// TIA Portal V16 export
// export: Created 2022-11-17T15:49:45.6262472Z, ExportSetting WithDefaults, DisplayName Totally Integrated Automation Portal, DisplayVersion V16 Update 6, DisplayName TIA Portal Version Control Interface, DisplayVersion V16 Update 2, DisplayName TIA Portal Openness, DisplayVersion V16 Update 6, DisplayName SINAMICS Startdrive Advanced, DisplayVersion V16 Update 5, DisplayName SINAMICS Startdrive G130, G150, S120, S150, SINAMICS MV, S210, DisplayVersion V16 Update 5, DisplayName SINAMICS Startdrive G110M, G120, G120C, G120D, G120P, G115D, DisplayVersion V16 Update 5, DisplayName STEP 7 Professional, DisplayVersion V16 Update 6, DisplayName STEP 7 Safety, DisplayVersion V16, DisplayName WinCC Advanced, DisplayVersion V16 Update 6
DATA_BLOCK "DB246_Program4"   // DB246
{ S7_Optimized_Access := 'FALSE' }
AUTHOR : Robopac
VERSION : 0.0
// stored: AutoNumber false, IsOnlyStoredInLoadMemory false, IsWriteProtectedInAS false
   VAR RETAIN
      Program4 { S7_SetPoint := 'True'} : "DatiProgramma";
   END_VAR
BEGIN
   Program4.Wrapping := TRUE;
   Program4.TopLenght := 500;
   Program4.TopRelease := 0;
   Program4.TopDown := 0;
   Program4.Top := 4;
   Program4.PressurePTime := 0;
   Program4.LifterTime := 0;
   Program4.RevOverContrast := 1;
   Program4.RopeEndCycle := 16#02;
   Program4.Spare4 := 16#01;
   Program4.RopeTime := 1500;
   Program4.RevOverClamp := 1;
   Program4.FilmForceFinalRev := 10;
   Program4.FilmPrestretchFinalRev := 100;
   Program4.ArmSpeed := 100;
   Program4.CarriageDown4Top := 500;
   Program4.TopDownTime := 1500;
   Program4.LapsUnderTop := 0;
   Program4.Spare6 := 0;
   Program4.Spare7 := 0;
   Program4.Spare8 := 0;
   Program4.Spare9 := 0;
   Program4.Spare10 := 0;
   Program4.Spare11 := 0;
   Program4.Spare12 := 0;
   Program4.Overlap0_1 := 0;
   Program4.Height1 := 130;
   Program4.Landmark1 := FALSE;
   Program4.Lifter1 := FALSE;
   Program4.SpareBit1H1 := FALSE;
   Program4.Airblower1 := TRUE;
   Program4.NextStep1 := TRUE;
   Program4.PressureP1 := TRUE;
   Program4.SpareByte2H1 := 16#00;
   Program4.Revolution1 := 1;
   Program4.RopeUnit1_1 := 16#01;
   Program4.RopeUnit1_2 := 16#01;
   Program4.FilmForce1 := 5;
   Program4.FilmPrestretch1 := 200;
   Program4.Spare3H1 := 0;
   Program4.Spare49 := 0;
   Program4.Spare50 := 0;
   Program4.Spare51 := 0;
   Program4.Spare52 := 0;
   Program4.Spare53 := 0;
   Program4.Overlap1_2 := 0;
   Program4.Height2 := 50;
   Program4.Landmark2 := FALSE;
   Program4.Lifter2 := FALSE;
   Program4.SpareBit1H2 := FALSE;
   Program4.Airblower2 := TRUE;
   Program4.NextStep2 := TRUE;
   Program4.PressureP2 := TRUE;
   Program4.SpareByte2H2 := 16#00;
   Program4.Revolution2 := 1;
   Program4.RopeUnit2_1 := 16#01;
   Program4.RopeUnit2_2 := 16#01;
   Program4.FilmForce2 := 20;
   Program4.FilmPrestretch2 := 200;
   Program4.Spare3H2 := 0;
   Program4.Spare54 := 0;
   Program4.Spare55 := 0;
   Program4.Spare56 := 0;
   Program4.Spare57 := 0;
   Program4.Spare58 := 0;
   Program4.Overlap2_3 := 100;
   Program4.Height3 := -50;
   Program4.Landmark3 := TRUE;
   Program4.Lifter3 := FALSE;
   Program4.SpareBit1H3 := FALSE;
   Program4.Airblower3 := TRUE;
   Program4.NextStep3 := TRUE;
   Program4.PressureP3 := TRUE;
   Program4.SpareByte2H3 := 16#00;
   Program4.Revolution3 := 2;
   Program4.RopeUnit3_1 := 16#01;
   Program4.RopeUnit3_2 := 16#01;
   Program4.FilmForce3 := 30;
   Program4.FilmPrestretch3 := 200;
   Program4.Spare3H3 := 0;
   Program4.Spare59 := 0;
   Program4.Spare60 := 0;
   Program4.Spare61 := 380;
   Program4.Spare62 := 2800;
   Program4.Spare63 := 0;
   Program4.Overlap3_4 := 100;
   Program4.Height4 := 100;
   Program4.Landmark4 := FALSE;
   Program4.Lifter4 := FALSE;
   Program4.SpareBit1H4 := FALSE;
   Program4.Airblower4 := TRUE;
   Program4.NextStep4 := TRUE;
   Program4.PressureP4 := TRUE;
   Program4.SpareByte2H4 := 16#00;
   Program4.Revolution4 := 3;
   Program4.RopeUnit4_1 := 16#02;
   Program4.RopeUnit4_2 := 16#02;
   Program4.FilmForce4 := 30;
   Program4.FilmPrestretch4 := 200;
   Program4.Spare3H4 := 0;
   Program4.Spare64 := 0;
   Program4.Spare65 := 0;
   Program4.Spare66 := 0;
   Program4.Spare67 := 0;
   Program4.Spare68 := 0;
   Program4.Overlap4_5 := 0;
   Program4.Height5 := 50;
   Program4.Landmark5 := FALSE;
   Program4.Lifter5 := FALSE;
   Program4.SpareBit1H5 := FALSE;
   Program4.Airblower5 := TRUE;
   Program4.NextStep5 := FALSE;
   Program4.PressureP5 := FALSE;
   Program4.SpareByte2H5 := 16#00;
   Program4.Revolution5 := 1;
   Program4.RopeUnit5_1 := 16#01;
   Program4.RopeUnit5_2 := 16#01;
   Program4.FilmForce5 := 30;
   Program4.FilmPrestretch5 := 200;
   Program4.Spare3H5 := 0;
   Program4.Spare69 := 0;
   Program4.Spare70 := 0;
   Program4.Spare71 := 0;
   Program4.Spare72 := 0;
   Program4.Spare73 := 0;
   Program4.Overlap5_6 := 100;
   Program4.Height6 := 50;
   Program4.Landmark6 := FALSE;
   Program4.Lifter6 := FALSE;
   Program4.SpareBit1H6 := FALSE;
   Program4.Airblower6 := TRUE;
   Program4.NextStep6 := FALSE;
   Program4.PressureP6 := FALSE;
   Program4.SpareByte2H6 := 16#00;
   Program4.Revolution6 := 2;
   Program4.RopeUnit6_1 := 16#02;
   Program4.RopeUnit6_2 := 16#01;
   Program4.FilmForce6 := 20;
   Program4.FilmPrestretch6 := 200;
   Program4.Spare3H6 := 0;
   Program4.Spare74 := 0;
   Program4.Spare75 := 0;
   Program4.Spare76 := 0;
   Program4.Spare77 := 0;
   Program4.Spare78 := 0;
   Program4.Overlap6_7 := 0;
   Program4.Height7 := 0;
   Program4.Landmark7 := FALSE;
   Program4.Lifter7 := FALSE;
   Program4.SpareBit1H7 := FALSE;
   Program4.Airblower7 := FALSE;
   Program4.NextStep7 := TRUE;
   Program4.PressureP7 := FALSE;
   Program4.SpareByte2H7 := 16#00;
   Program4.Revolution7 := 1;
   Program4.RopeUnit7_1 := 16#01;
   Program4.RopeUnit7_2 := 16#01;
   Program4.FilmForce7 := 0;
   Program4.FilmPrestretch7 := 100;
   Program4.Spare3H7 := 0;
   Program4.Spare79 := 0;
   Program4.Spare80 := 0;
   Program4.Spare81 := 0;
   Program4.Spare82 := 0;
   Program4.Spare83 := 0;
   Program4.Overlap7_8 := 0;
   Program4.Height8 := 0;
   Program4.Landmark8 := FALSE;
   Program4.Lifter8 := FALSE;
   Program4.SpareBit1H8 := FALSE;
   Program4.Airblower8 := FALSE;
   Program4.NextStep8 := TRUE;
   Program4.PressureP8 := FALSE;
   Program4.SpareByte2H8 := 16#00;
   Program4.Revolution8 := 1;
   Program4.RopeUnit8_1 := 16#01;
   Program4.RopeUnit8_2 := 16#01;
   Program4.FilmForce8 := 0;
   Program4.FilmPrestretch8 := 100;
   Program4.Spare3H8 := 0;
   Program4.Spare84 := 0;
   Program4.Spare85 := 0;
   Program4.Spare86 := 0;
   Program4.Spare87 := 0;
   Program4.Spare88 := 0;
   Program4.Overlap8_9 := 0;
   Program4.Height9 := 0;
   Program4.Landmark9 := FALSE;
   Program4.Lifter9 := FALSE;
   Program4.SpareBit1H9 := FALSE;
   Program4.Airblower9 := FALSE;
   Program4.NextStep9 := TRUE;
   Program4.PressureP9 := FALSE;
   Program4.SpareByte2H9 := 16#00;
   Program4.Revolution9 := 1;
   Program4.RopeUnit9_1 := 16#01;
   Program4.RopeUnit9_2 := 16#01;
   Program4.FilmForce9 := 0;
   Program4.FilmPrestretch9 := 100;
   Program4.Spare3H9 := 0;
   Program4.Spare89 := 0;
   Program4.Spare90 := 0;
   Program4.Spare91 := 0;
   Program4.Spare92 := 0;
   Program4.Spare93 := 0;
   Program4.Overlap9_10 := 0;
   Program4.Height10 := 0;
   Program4.Landmark10 := FALSE;
   Program4.Lifter10 := FALSE;
   Program4.SpareBit1H10 := FALSE;
   Program4.Airblower10 := FALSE;
   Program4.NextStep10 := FALSE;
   Program4.PressureP10 := FALSE;
   Program4.SpareByte2H10 := 16#00;
   Program4.Revolution10 := 1;
   Program4.RopeUnit10_1 := 16#01;
   Program4.RopeUnit10_2 := 16#01;
   Program4.FilmForce10 := 0;
   Program4.FilmPrestretch10 := 100;
   Program4.Spare3H10 := 0;
   Program4.Spare94 := 0;
   Program4.Spare95 := 0;
   Program4.Spare96 := 0;
   Program4.Spare97 := 0;
   Program4.Spare98 := 0;
   Program4.Overlap10_11 := 0;
   Program4.Height11 := 0;
   Program4.Landmark11 := FALSE;
   Program4.Lifter11 := FALSE;
   Program4.SpareBit1H11 := FALSE;
   Program4.Airblower11 := FALSE;
   Program4.NextStep11 := TRUE;
   Program4.PressureP11 := FALSE;
   Program4.SpareByte2H11 := 16#00;
   Program4.Revolution11 := 1;
   Program4.RopeUnit11_1 := 16#01;
   Program4.RopeUnit11_2 := 16#01;
   Program4.FilmForce11 := 0;
   Program4.FilmPrestretch11 := 100;
   Program4.Spare3H11 := 0;
   Program4.Spare99 := 0;
   Program4.Spare100 := 0;
   Program4.Spare101 := 0;
   Program4.Spare102 := 0;
   Program4.Spare103 := 0;
   Program4.Overlap11_12 := 0;
   Program4.Height12 := 0;
   Program4.Landmark12 := FALSE;
   Program4.Lifter12 := FALSE;
   Program4.SpareBit1H12 := FALSE;
   Program4.Airblower12 := FALSE;
   Program4.NextStep12 := FALSE;
   Program4.PressureP12 := FALSE;
   Program4.SpareByte2H12 := 16#00;
   Program4.Revolution12 := 1;
   Program4.RopeUnit12_1 := 16#01;
   Program4.RopeUnit12_2 := 16#01;
   Program4.FilmForce12 := 0;
   Program4.FilmPrestretch12 := 100;
   Program4.Spare3H12 := 0;
   Program4.Spare104 := 0;
   Program4.Spare105 := 0;
   Program4.Spare106 := 0;
   Program4.Spare107 := 0;
   Program4.Spare108 := 0;
END_DATA_BLOCK
